FUNCTION_BLOCK FB_Observer_BOOL EXTENDS FB_AbstractObserver
VAR
    _bVal:      BOOL;
END_VAR

PROPERTY bValue : BOOL
GET
bValue := THIS^._bVal;
END_GET
END_PROPERTY

METHOD FB_init : BOOL
VAR_INPUT
	bInitRetains : BOOL; // if TRUE, the retain variables are initialized (warm start / cold start)
	bInCopyCode : BOOL;  // if TRUE, the instance afterwards gets moved into the copy code (online change)
END_VAR
THIS^._nTypeClass := __SYSTEM.TYPE_CLASS.TYPE_BOOL;
THIS^._pVal := ADR(THIS^._bVal);
THIS^._nSize := SIZEOF(THIS^._bVal);
END_METHOD

END_FUNCTION_BLOCK

(* stored: Version 1.1.0.1, ProductVersion 3.1.4024.12
   POU FB_Observer_BOOL: Id {b69e048a-892f-4809-8b52-c7b077bb4215}, SpecialFunc None
   Property bValue: Id {a4508b65-b06d-49ac-ade8-4e663f660e99}
   Get Get: Id {98ab5782-160e-45c0-a473-069f68784c18}
   Method FB_init: Id {5a187cdb-5624-4c83-96a8-6a6f18ce82cc} *)
